// Mitsubishi GX Works2 project: z01   PLC: Q02/Q02H

PROGRAM MAIN
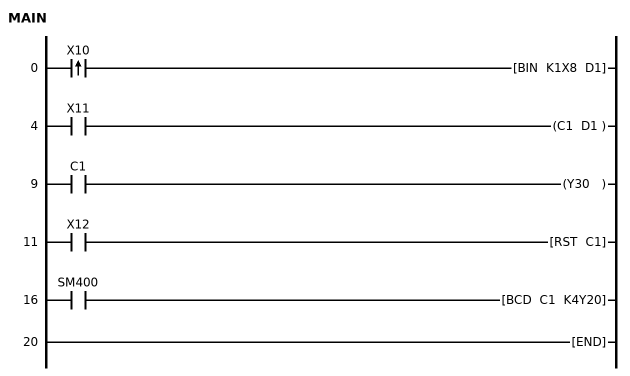
0     LDP     X10
      BIN     K1X8 D1
4     LD      X11
      OUT     C1 D1
9     LD      C1
      OUT     Y30
11    LD      X12
      RST     C1
16    LD      SM400
      BCD     C1 K4Y20
20    END
END_PROGRAM
